// TwinCAT 3 PLC project PRG_Test_Periphery
// Company: RafalOS
// ProgramVersion: 3.1.4024.0
// libraries:
//   B_Actuator, * (RafalOS)
//   B_ActuatorDecorator, * (RafalOS)
//   B_Base, * (RafalOS)
//   B_IO, * (RafalOS)
//   B_IODecorator, * (RafalOS)
//   Tc2_DataExchange, * (Beckhoff Automation GmbH)
//   Tc2_Standard, * (Beckhoff Automation GmbH)
//   Tc2_System, * (Beckhoff Automation GmbH)
//   Tc3_Module, * (Beckhoff Automation GmbH)
//   TcUnit, * (www.tcunit.org)
// project tree:
//   GVLs/ GVL_Actuator.TcGVL, GVL_Decorators.TcGVL, GVL_Variable.TcGVL (not stored)
//   / PlcTask.TcTTO (not stored)
//   POUs/ FB_ActuatorTest.TcPOU, FB_ButtonTest.TcPOU, FB_ElectroValveTest.TcPOU, FB_LampBlinkingTest.TcPOU (not stored), FB_Sensor_DecoratorTestTest.TcPOU, FB_SensorTest.TcPOU (not stored), FB_Actuator_TestDecoratorWithoutTimeTest.TcPOU (not stored), FB_Actuator_TestDecoratorWithTimeTest.TcPOU
//   TESTs/ PRG_Test.TcPOU (not stored)

// ---- GVLs/GVL_Actuator.TcGVL
{attribute 'qualified_only'}
VAR_GLOBAL
	flSS1						: FB_BaseFlag;
	flSTO						: FB_BaseFlag;
	fbLogger					: FB_BaseLogger;
	fbTime						: FB_BaseTime;
	fbLocaciotn					: FB_BaseLocation;	
	stCommonData				: ST_BaseCommonData;

	senActuatorStart			: FB_Sensor_NO;
	senActuatorEnd				: FB_Sensor_NO;
	evActuator					: FB_Electrovalve_5on3_2Coil_Vented;
	
	actActuator					: FB_Actuator (
									senStart	:= senActuatorStart,
	                                senEnd		:= senActuatorEnd,
	                                evControl	:= evActuator
								);
								
END_VAR

// ---- GVLs/GVL_Decorators.TcGVL
{attribute 'qualified_only'}
VAR_GLOBAL
	senNO				: FB_Sensor_NO;
	senNC				: FB_Sensor_NC;
	senNO_2inRow		: FB_Sensor_NO_2InRow;
	
	senNO_TestDecorator			: FB_Sensor_NO_TestDecorator (fbToDecorate := senNO);
	senNC_TestDecorator			: FB_Sensor_NC_TestDecorator (fbToDecorate := senNC);
	senNO_2inRow_TestDecorator	: FB_Sensor_NO_2InRow_TestDecorator (fbToDecorate := senNO_2inRow);
	
	
	senActuator1Start		: FB_Sensor_NO;
	senActuator1End			: FB_Sensor_NO;
	evActuator1				: FB_Electrovalve_5on2_1Coil;

	senActuator1Start_TestCecorator		: FB_Sensor_NO_TestDecorator (fbToDecorate := senActuator1Start);
	senActuator1End_TestDecorator		: FB_Sensor_NO_TestDecorator (fbToDecorate := senActuator1End);
	
	actActuator1			: FB_Actuator (
								senStart	:= senActuator1Start_TestCecorator,
								senEnd		:= senActuator1End_TestDecorator,
								evControl	:= evActuator1
							);
	
	actActuator1_TestWithoutTimeDecorator	: FB_Actuator_TestWithoutTimeDecorator (
											fbToDecorate	:= actActuator1,
											actActuator		:= actActuator1,
											senStart		:= senActuator1Start_TestCecorator,
											senEnd			:= senActuator1End_TestDecorator
										);
	

	actActuator1_TestWithTimeDecorator	: FB_Actuator_TestWithTimeDecorator (
											fbToDecorate	:= actActuator1,
											actActuator		:= actActuator1,
											senStart		:= senActuator1Start_TestCecorator,
											senEnd			:= senActuator1End_TestDecorator
										);
	flSS1						: FB_BaseFlag;
	flSTO						: FB_BaseFlag;
	fbLogger					: FB_BaseLogger;
	fbTime						: FB_BaseTime;
	fbLocaciotn					: FB_BaseLocation;	
	stCommonData				: ST_BaseCommonData;
	
END_VAR

// ---- POUs/FB_ActuatorTest.TcPOU
FUNCTION_BLOCK FB_ActuatorTest EXTENDS TcUnit.FB_TestSuite
VAR

END_VAR


GVL_Actuator.actActuator.ExecuteEveryCycle_Test ();
GVL_Actuator.actActuator.ExecuteEveryCycle_Operation ();
GVL_Actuator.actActuator.ExecuteEveryCycle_Status ();
GVL_Actuator.actActuator.ExecuteEveryCycle_Error ();

T01_Parameter ();
T02_TestMove ();

METHOD PROTECTED T01_Parameter
VAR_INPUT
END_VAR

VAR
	uiWynik: UINT;
	rWynik: REAL;
END_VAR
IF (TcUnit.TEST_ORDERED ('T01_Parameter')) THEN
	GVL_Actuator.stCommonData.itfLocaciotn	:= GVL_Actuator.fbLocaciotn;
	GVL_Actuator.stCommonData.itfLogger		:= GVL_Actuator.fbLogger;
	GVL_Actuator.stCommonData.itfTime		:= GVL_Actuator.fbTime;
	GVL_Actuator.actActuator.LinkCommonData (stCommonData := GVL_Actuator.stCommonData);
	GVL_Actuator.actActuator.LinkSS1 (fbSS1	:= GVL_Actuator.flSS1);
	GVL_Actuator.actActuator.LinkSTO (fbSTO	:= GVL_Actuator.flSTO);
	
	GVL_Actuator.flSS1.SetFlag (bState := TRUE);
	GVL_Actuator.flSTO.SetFlag (bState := TRUE);

	GVL_Actuator.actActuator.ParametersCreate ();
	
	uiWynik		:= GVL_Actuator.actActuator.ParameterGetNumberOfAdded ();
	AssertEquals_UINT (Expected := 2, Actual := uiWynik, Message := 'T01 - Bledna ilosc parametrow');
	rWynik		:= GVL_Actuator.actActuator.ParameterGetValue (uiNumber := 1);
	AssertEquals_REAL (Expected := 100, Actual := rWynik, Delta := 0, Message := 'T02 - bladna wartosc');
	rWynik		:= GVL_Actuator.actActuator.ParameterGetValue (uiNumber := 2);
	AssertEquals_REAL (Expected := 100, Actual := rWynik, Delta := 0, Message := 'T03 - bladna wartosc');

	GVL_Actuator.actActuator.ParameterCorrectValue (uiNumber := 1, rValue := 1000);
	GVL_Actuator.actActuator.ParameterCorrectValue (uiNumber := 2, rValue := 1000);
	rWynik		:= GVL_Actuator.actActuator.ParameterGetValue (uiNumber := 1);
	AssertEquals_REAL (Expected := 1000, Actual := rWynik, Delta := 0, Message := 'T04 - bladna wartosc');
	rWynik		:= GVL_Actuator.actActuator.ParameterGetValue (uiNumber := 2);
	AssertEquals_REAL (Expected := 1000, Actual := rWynik, Delta := 0, Message := 'T05 - bladna wartosc');

	GVL_Actuator.actActuator.ParameterCorrectValue (uiNumber := 1, rValue := 100);
	GVL_Actuator.actActuator.ParameterCorrectValue (uiNumber := 2, rValue := 100);
	
	
	TcUnit.TEST_FINISHED ();
END_IF
END_METHOD

METHOD PRIVATE T02_TestMove
VAR_INST
	iStep			: int;
END_VAR
IF (TcUnit.TEST_ORDERED ('T02_TestMove')) THEN
	CASE iStep OF
	0	:
		GVL_Actuator.actActuator.PowerTurnOn ();
		iStep		:= iStep + 10;
	10	:
		IF (GVL_Actuator.actActuator.PowerTurnOnDone ()) THEN
			iStep	:= iStep + 10;
		END_IF
	20	:
		GVL_Actuator.actActuator.MoveToStart ();
		iStep		:= iStep + 10;
	30	:
		AssertTrue (Condition := GVL_Actuator.actActuator.MovingToStartBusy (), Message := 'S30 - T01 - nie uruchomione przesuwanie');
		AssertFalse (Condition :=GVL_Actuator.actActuator.MovingToStartStatus (), Message := 'S30 - T02 - Bledny status');
		iStep		:= iStep + 10;
	40	:
		GVL_Variable.bValueToSave	:= TRUE;
		GVL_Variable.sData			:= 'GVL_Actuator.senActuatorStart.bContact';
		GVL_Variable.bSave			:= TRUE;
		iStep		:= iStep + 10;
	50	:
		IF (NOT GVL_Variable.bSaved) THEN
			GVL_Variable.bSave		:= FALSE;
			iStep	:= iStep + 10;
		END_IF
	60	:
		AssertFalse (Condition := GVL_Actuator.actActuator.MovingToStartBusy (), Message := 'S60 - T01 - nie zakonczone przesuwanie');
		AssertTrue (Condition := GVL_Actuator.actActuator.MovingToStartStatus (), Message := 'S60 - T02 - Bledny status');
		AssertTrue (Condition := GVL_Actuator.senActuatorStart.IsActive (), Message := 'S60 - T03 - Bledny stan czujnika');
	
		iStep		:= 1000;
	1000	:
		TcUnit.TEST_FINISHED ();
	END_CASE
END_IF
END_METHOD

END_FUNCTION_BLOCK

// ---- POUs/FB_ButtonTest.TcPOU
FUNCTION_BLOCK FB_ButtonTest EXTENDS TcUnit.FB_TestSuite
VAR
END_VAR

T01_Przycisk_NC ();
T02_Przycisk_NO ();
T03_PrzyciskNC_Impuls ();
T04_PrzyciskNO_Impuls ();

METHOD PROTECTED T01_Przycisk_NC
IF (TcUnit.TEST_ORDERED ('T01_Przycisk_NC')) THEN 
	//Przycisk nie jest nacisniety
	WRITE_PROTECTED_BOOL (ADR (GVL_Variable.fbButton_NC.bcontact), TRUE);
	//odczyt
	AssertEquals_BOOL (Actual := GVL_Variable.fbButton_NC.IsPressed (), Expected := FALSE, Message := '1 - Bledny odczyt styku');
	//Przycisk jest nacisniety
	WRITE_PROTECTED_BOOL (ADR (GVL_Variable.fbButton_NC.bContact), FALSE);
	//odczyt
	AssertEquals_BOOL (Actual := GVL_Variable.fbButton_NC.IsPressed (), Expected := TRUE, Message := '2 - Bledny odczyt styku');
	
	TcUnit.TEST_FINISHED ();
END_IF
END_METHOD

METHOD PROTECTED T02_Przycisk_NO
VAR
	bCzyNaciskniety: BOOL;
	bCzySwieci: BOOL;
END_VAR
IF (TcUnit.TEST_ORDERED ('T02_Przycisk_NO')) THEN 
	//Przycisk nie jest nacisniety
	WRITE_PROTECTED_BOOL (ADR (GVL_Variable.fbButton_NO.bContact), FALSE);
	//odczyt
	AssertEquals_BOOL (Actual := GVL_Variable.fbButton_NO.IsPressed (), Expected := FALSE, Message := '1 - Bledny odczyt styku');
	//Przycisk jest nacisniety
	WRITE_PROTECTED_BOOL (ADR (GVL_Variable.fbButton_NO.bContact), TRUE);
	//odczyt
	AssertEquals_BOOL (Actual := GVL_Variable.fbButton_NO.IsPressed (), Expected := TRUE, Message := '2 - Bledny odczyt styku');

	TcUnit.TEST_FINISHED ();
END_IF
END_METHOD

METHOD PROTECTED T03_PrzyciskNC_Impuls
VAR_INST
	iKrok: INT;
END_VAR
IF (TcUnit.TEST_ORDERED ('T03_PrzyciskNC_Impuls')) THEN
	CASE iKrok OF
		0	: 
			WRITE_PROTECTED_BOOL (Ptr := ADR(GVL_Variable.fbButton_NC.bContact), Value := FALSE);
			iKrok		:= 10;
		10	:
			AssertTrue (Condition := GVL_Variable.fbButton_NC.GetRisingEdgePressed (), Message := '10 - Bledny odczyt styku');
			iKrok		:= 20;
		20	:
			AssertFalse (Condition := GVL_Variable.fbButton_NC.GetRisingEdgePressed (), Message := '20 - Bledny odczyt styku');
			iKrok		:= 30;
		30	:
			WRITE_PROTECTED_BOOL (Ptr := ADR(GVL_Variable.fbButton_NC.bContact), Value := TRUE);
			iKrok		:= 40;
		40	:
			AssertFalse (Condition := GVL_Variable.fbButton_NC.GetRisingEdgePressed (), Message := '40 - Bledny odczyt styku');
			iKrok		:= 500;
		500	:
			TcUnit.TEST_FINISHED ();
	END_CASE	
END_IF
END_METHOD

METHOD PROTECTED T04_PrzyciskNO_Impuls
VAR_INST
	iKrok: INT;
END_VAR
IF (TcUnit.TEST_ORDERED ('T04_PrzyciskNO_Impuls')) THEN
	CASE iKrok OF
		0	: 
			WRITE_PROTECTED_BOOL (Ptr := ADR(GVL_Variable.fbButton_NO.bContact), Value := TRUE);
			iKrok		:= 10;
		10	:
			AssertTrue (Condition := GVL_Variable.fbButton_NO.GetRisingEdgePressed (), Message := '10 - Bledny odczyt styku');
			iKrok		:= 20;
		20	:
			AssertFalse (Condition := GVL_Variable.fbButton_NO.GetRisingEdgePressed (), Message := '20 - Bledny odczyt styku');
			iKrok		:= 30;
		30	:
			WRITE_PROTECTED_BOOL (Ptr := ADR(GVL_Variable.fbButton_NO.bContact), Value := FALSE);
			iKrok 		:= 35;
		35	:
			AssertFalse (Condition := GVL_Variable.fbButton_NO.GetRisingEdgePressed (), Message := '35 - Bledny odczyt styku');
			iKrok		:= 40;
		40	:
			WRITE_PROTECTED_BOOL (Ptr := ADR(GVL_Variable.fbButton_NO.bContact), Value := TRUE);
			AssertTrue (Condition := GVL_Variable.fbButton_NO.IsPressed (), Message := '40a - Bledny odczyt styku');
			iKrok 		:= ikrok + 10;
		50	:
			AssertTrue (Condition := GVL_Variable.fbButton_NO.GetRisingEdgePressed (), Message := '50a - Bledny odczyt styku');
			iKrok 		:= ikrok + 10;
		60	:
			AssertFalse (Condition := GVL_Variable.fbButton_NO.GetRisingEdgePressed (), Message := '60b - Bledny odczyt styku');
			iKrok 		:= ikrok + 10;
		70	:
			WRITE_PROTECTED_BOOL (Ptr := ADR(GVL_Variable.fbButton_NO.bContact), Value := FALSE);
			iKrok 		:= ikrok + 10;
		80	:
			AssertFalse (Condition := GVL_Variable.fbButton_NO.GetRisingEdgePressed (), Message := '80c - Bledny odczyt styku');
			iKrok		:= 500;
		500	:
			TcUnit.TEST_FINISHED ();
	END_CASE
	
END_IF
END_METHOD

END_FUNCTION_BLOCK

// ---- POUs/FB_ElectroValveTest.TcPOU
FUNCTION_BLOCK FB_ElectroValveTest EXTENDS TcUnit.FB_TestSuite
VAR
END_VAR

T01_El3Na2_NC ();
T02_El3Na2_NO ();
T03_El5Na2_1C ();
T04_El5Na2_2C ();
T05_El5Na3_2C_odp ();
T06_El5Na3_2C_zap ();

METHOD PROTECTED T01_El3Na2_NC
VAR_INPUT
END_VAR
IF (TcUnit.TEST_ORDERED ('T01_El3Na2_NC')) THEN
	GVL_Variable.ev3on2_NC.Contol (eAction 	:= E_ElectrovalveAction.e_EV_OUT4_Active);
	AssertTrue (
		Condition							:= GVL_Variable.ev3on2_NC.bCoilA,
		Message								:= 'Test 1 - blad przelaczania'
	);
	GVL_Variable.ev3on2_NC.Contol (eAction 	:= E_ElectrovalveAction.e_EV_Out4_Deactive);
	AssertFalse (
		Condition							:= GVL_Variable.ev3on2_NC.bCoilA,
		Message								:= 'Test 2 - blad przelaczania'
	);
	GVL_Variable.ev3on2_NC.Contol (eAction 	:= E_ElectrovalveAction.e_EV_OUT4_Active);
	AssertTrue (
		Condition							:= GVL_Variable.ev3on2_NC.bCoilA,
		Message								:= 'Test 3 - blad przelaczania'
	);
	GVL_Variable.ev3on2_NC.Contol (eAction 	:= E_ElectrovalveAction.e_EV_Reset);
	AssertFalse (
		Condition							:= GVL_Variable.ev3on2_NC.bCoilA,
		Message								:= 'Test 4 - blad przelaczania'
	);
	

	TcUnit.TEST_FINISHED ();
END_IF
END_METHOD

METHOD PROTECTED T02_El3Na2_NO
VAR_INPUT
END_VAR
IF (TcUnit.TEST_ORDERED ('T02_El3Na2_NO')) THEN
	GVL_Variable.ev3on2_NC.Contol (eAction 	:= E_ElectrovalveAction.e_EV_OUT4_Active);
	AssertTrue (
		Condition							:= GVL_Variable.ev3on2_NC.bCoilA,
		Message								:= 'Test 1 - blad przelaczania'
	);
	GVL_Variable.ev3on2_NC.Contol (eAction 	:= E_ElectrovalveAction.e_EV_Out4_Deactive);
	AssertFalse (
		Condition							:= GVL_Variable.ev3on2_NC.bCoilA,
		Message								:= 'Test 2 - blad przelaczania'
	);
	GVL_Variable.ev3on2_NC.Contol (eAction 	:= E_ElectrovalveAction.e_EV_OUT4_Active);
	AssertTrue (
		Condition							:= GVL_Variable.ev3on2_NC.bCoilA,
		Message								:= 'Test 3 - blad przelaczania'
	);
	GVL_Variable.ev3on2_NC.Contol (eAction 	:= E_ElectrovalveAction.e_EV_Reset);
	AssertFalse (
		Condition							:= GVL_Variable.ev3on2_NC.bCoilA,
		Message								:= 'Test 4 - blad przelaczania'
	);
	

	TcUnit.TEST_FINISHED ();
END_IF
END_METHOD

METHOD PROTECTED T03_El5Na2_1C
VAR_INPUT
END_VAR
IF (TcUnit.TEST_ORDERED ('T03_El5Na2_1C')) THEN
	GVL_Variable.ev5on2_1C.Contol (eAction 	:= E_ElectrovalveAction.e_EV_OUT4_Active);
	AssertTrue (
		Condition							:= GVL_Variable.ev5on2_1C.bCoilA,
		Message								:= 'Test 1 - blad przelaczania'
	);
	
	GVL_Variable.ev5on2_1C.Contol (eAction 	:= E_ElectrovalveAction.e_EV_Out4_Deactive);
	AssertFalse (
		Condition							:= GVL_Variable.ev5on2_1C.bCoilA,
		Message								:= 'Test 2 - blad przelaczania'
	);
	
	GVL_Variable.ev5on2_1C.Contol (eAction 	:= E_ElectrovalveAction.e_EV_ToStart);
	AssertFalse (
		Condition							:= GVL_Variable.ev5on2_1C.bCoilA,
		Message								:= 'Test 1 - blad przelaczania'
	);

	GVL_Variable.ev5on2_1C.Contol (eAction 	:= E_ElectrovalveAction.e_EV_ToEnd);
	AssertTrue (
		Condition							:= GVL_Variable.ev5on2_1C.bCoilA,
		Message								:= 'Test 2 - blad przelaczania'
	);
	

	TcUnit.TEST_FINISHED ();
END_IF
END_METHOD

METHOD PROTECTED T04_El5Na2_2C
VAR_INPUT
END_VAR
IF (TcUnit.TEST_ORDERED ('T04_El5Na2_2C')) THEN
	GVL_Variable.ev5on2_2C.Contol (eAction 	:= E_ElectrovalveAction.e_EV_OUT4_Active);
	AssertTrue (
		Condition							:= GVL_Variable.ev5on2_2C.bCoilA,
		Message								:= 'Test 1A - Blad przelaczania'
	);
	Assertfalse (
		Condition							:= GVL_Variable.ev5on2_2C.bCoilB,
		Message								:= 'Test 1B - Blad przelaczania'
	);
//
	GVL_Variable.ev5on2_2C.Contol (eAction 	:= E_ElectrovalveAction.e_EV_Out2_Active);
	AssertFalse (
		Condition							:= GVL_Variable.ev5on2_2C.bCoilA,
		Message								:= 'Test 2A - Blad przelaczania'
	);
	AssertTrue (
		Condition							:= GVL_Variable.ev5on2_2C.bCoilB,
		Message								:= 'Test 2B - Blad przelaczania'
	);
//
	GVL_Variable.ev5on2_2C.Contol (eAction 	:= E_ElectrovalveAction.e_EV_ToEnd);
	AssertTrue (
		Condition							:= GVL_Variable.ev5on2_2C.bCoilA,
		Message								:= 'Test 3A - Blad przelaczania'
	);
	Assertfalse (
		Condition							:= GVL_Variable.ev5on2_2C.bCoilB,
		Message								:= 'Test 3B - Blad przelaczania'
	);
//
	GVL_Variable.ev5on2_2C.Contol (eAction 	:= E_ElectrovalveAction.e_EV_ToStart);
	AssertFalse (
		Condition							:= GVL_Variable.ev5on2_2C.bCoilA,
		Message								:= 'Test 4A - Blad przelaczania'
	);
	AssertTrue (
		Condition							:= GVL_Variable.ev5on2_2C.bCoilB,
		Message								:= 'Test 4B - Blad przelaczania'
	);
//
	GVL_Variable.ev5on2_2C.Contol (eAction 	:= E_ElectrovalveAction.e_EV_Reset);
	AssertFalse (
		Condition							:= GVL_Variable.ev5on2_2C.bCoilA,
		Message								:= 'Test 5A - Blad przelaczania'
	);
	AssertFalse (
		Condition							:= GVL_Variable.ev5on2_2C.bCoilB,
		Message								:= 'Test 5B - Blad przelaczania'
	);
	TcUnit.TEST_FINISHED ();
END_IF
END_METHOD

METHOD PROTECTED T05_El5Na3_2C_odp
VAR_INPUT
END_VAR
IF (TcUnit.TEST_ORDERED ('T05_El5Na3_2C_odp')) THEN
	GVL_Variable.ev5on3_2C_ven.Contol (eAction 	:= E_ElectrovalveAction.e_EV_OUT4_Active);
	AssertTrue (
		Condition							:= GVL_Variable.ev5on3_2C_ven.bCoilA,
		Message								:= 'Test 1A - Blad przelaczania'
	);
//
	GVL_Variable.ev5on3_2C_ven.Contol (eAction 	:= E_ElectrovalveAction.e_EV_Out2_Active);
	AssertTrue (
		Condition							:= GVL_Variable.ev5on3_2C_ven.bCoilB,
		Message								:= 'Test 2B - Blad przelaczania'
	);
//
	GVL_Variable.ev5on3_2C_ven.Contol (eAction 	:= E_ElectrovalveAction.e_EV_Reset);
	AssertFalse (
		Condition							:= GVL_Variable.ev5on3_2C_ven.bCoilA,
		Message								:= 'Test 3A - Blad przelaczania'
	);
	AssertFalse (
		Condition							:= GVL_Variable.ev5on3_2C_ven.bCoilB,
		Message								:= 'Test 3B - Blad przelaczania'
	);
//
	GVL_Variable.ev5on3_2C_ven.Contol (eAction 	:= E_ElectrovalveAction.e_EV_ToStart);
	AssertFalse (
		Condition							:= GVL_Variable.ev5on3_2C_ven.bCoilA,
		Message								:= 'Test 4A - Blad przelaczania'
	);
	AssertTrue (
		Condition							:= GVL_Variable.ev5on3_2C_ven.bCoilB,
		Message								:= 'Test 4B - Blad przelaczania'
	);
//
	GVL_Variable.ev5on3_2C_ven.Contol (eAction 	:= E_ElectrovalveAction.e_EV_ToEnd);
	AssertTrue (
		Condition							:= GVL_Variable.ev5on3_2C_ven.bCoilA,
		Message								:= 'Test 5A - Blad przelaczania'
	);
	Assertfalse (
		Condition							:= GVL_Variable.ev5on3_2C_ven.bCoilB,
		Message								:= 'Test 5B - Blad przelaczania'
	);
//
	GVL_Variable.ev5on3_2C_ven.Contol (eAction 	:= E_ElectrovalveAction.e_EV_Stop);
	AssertTrue (
		Condition							:= GVL_Variable.ev5on3_2C_ven.bCoilA,
		Message								:= 'Test 6A - Blad przelaczania'
	);
	AssertTrue (
		Condition							:= GVL_Variable.ev5on3_2C_ven.bCoilB,
		Message								:= 'Test 6B - Blad przelaczania'
	);
	
	TcUnit.TEST_FINISHED ();
END_IF
END_METHOD

METHOD PROTECTED T06_El5Na3_2C_zap
VAR_INPUT
END_VAR
IF (TcUnit.TEST_ORDERED ('T06_El5Na3_2C_zap')) THEN
	GVL_Variable.ev5on3_2C_inf.Contol (eAction 	:= E_ElectrovalveAction.e_EV_Out4_Deactive);
	AssertTrue (
		Condition							:= GVL_Variable.ev5on3_2C_inf.bCoilA,
		Message								:= 'Test 1A - Blad przelaczania'
	);
//
	GVL_Variable.ev5on3_2C_inf.Contol (eAction 	:= E_ElectrovalveAction.e_EV_Out2_Deactive);
	AssertTrue (
		Condition							:= GVL_Variable.ev5on3_2C_inf.bCoilB,
		Message								:= 'Test 2B - Blad przelaczania'
	);
//
	GVL_Variable.ev5on3_2C_inf.Contol (eAction 	:= E_ElectrovalveAction.e_EV_Reset);
	AssertFalse (
		Condition							:= GVL_Variable.ev5on3_2C_inf.bCoilA,
		Message								:= 'Test 3A - Blad przelaczania'
	);
	AssertFalse (
		Condition							:= GVL_Variable.ev5on3_2C_inf.bCoilB,
		Message								:= 'Test 3B - Blad przelaczania'
	);
//
	GVL_Variable.ev5on3_2C_inf.Contol (eAction 	:= E_ElectrovalveAction.e_EV_ToStart);
	AssertTrue (
		Condition							:= GVL_Variable.ev5on3_2C_inf.bCoilA,
		Message								:= 'Test 4A - Blad przelaczania'
	);
	AssertFalse (
		Condition							:= GVL_Variable.ev5on3_2C_inf.bCoilB,
		Message								:= 'Test 4B - Blad przelaczania'
	);
//
	GVL_Variable.ev5on3_2C_inf.Contol (eAction 	:= E_ElectrovalveAction.e_EV_ToEnd);
	AssertFalse (
		Condition							:= GVL_Variable.ev5on3_2C_inf.bCoilA,
		Message								:= 'Test 5A - Blad przelaczania'
	);
	AssertTrue (
		Condition							:= GVL_Variable.ev5on3_2C_inf.bCoilB,
		Message								:= 'Test 5B - Blad przelaczania'
	);
//
	GVL_Variable.ev5on3_2C_inf.Contol (eAction 	:= E_ElectrovalveAction.e_EV_Stop);
	AssertFalse (
		Condition							:= GVL_Variable.ev5on3_2C_inf.bCoilA,
		Message								:= 'Test 6A - Blad przelaczania'
	);
	AssertFalse (
		Condition							:= GVL_Variable.ev5on3_2C_inf.bCoilB,
		Message								:= 'Test 6B - Blad przelaczania'
	);
	
	TcUnit.TEST_FINISHED ();
END_IF
END_METHOD

END_FUNCTION_BLOCK

// ---- POUs/FB_Sensor_DecoratorTestTest.TcPOU
FUNCTION_BLOCK FB_Sensor_DecoratorTestTest EXTENDS TcUnit.FB_TestSuite
VAR

END_VAR


T01_TestCzujnikNC ();
T02_TestCzujnikNO ();
T03_TestCzujnikNO_Szereg ();

METHOD PROTECTED T01_TestCzujnikNC
VAR_INST
	iKrok		: INT;
END_VAR
IF (TcUnit.TEST_ORDERED ('T01_TestCzujnikNC')) THEN
	GVL_Decorators.senNC_TestDecorator.SetContact (bIN := TRUE);
	AssertFalse (Condition := GVL_Decorators.senNC_TestDecorator.IsActive (), Message := 'T11 - bledny stan');
	GVL_Decorators.senNC_TestDecorator.SetContact (bIN := FALSE);
	AssertTrue (Condition := GVL_Decorators.senNC_TestDecorator.IsActive (), Message := 'T12 - bledny stan');
	GVL_Decorators.senNC_TestDecorator.SetContact (bIN := TRUE);
	AssertFalse (Condition := GVL_Decorators.senNC_TestDecorator.IsActive (), Message := 'T13 - bledny stan');
	
	TcUnit.TEST_FINISHED ();
END_IF
END_METHOD

METHOD PROTECTED T02_TestCzujnikNO
VAR_INST
	iKrok		: INT;
END_VAR
IF (TcUnit.TEST_ORDERED ('T02_TestCzujnikNO')) THEN
	GVL_Decorators.senNO_TestDecorator.SetContact (bIN := FALSE);
	AssertFalse (Condition := GVL_Decorators.senNo_TestDecorator.IsActive (), Message := 'T11 - bledny stan');
	GVL_Decorators.senNO_TestDecorator.SetContact (bIN := TRUE);
	AssertTrue (Condition := GVL_Decorators.senNO_TestDecorator.IsActive (), Message := 'T12 - bledny stan');
	GVL_Decorators.senNO_TestDecorator.SetContact (bIN := FALSE);
	AssertFalse (Condition := GVL_Decorators.senNO_TestDecorator.IsActive (), Message := 'T13 - bledny stan');

	TcUnit.TEST_FINISHED ();
END_IF
END_METHOD

METHOD PROTECTED T03_TestCzujnikNO_Szereg
VAR_INST
	ikrok			: int;
END_VAR
IF (TcUnit.TEST_ORDERED ('T03_TestCzujnikNO_Szereg')) THEN
	GVL_Decorators.senNO_2inRow_TestDecorator.SetContact (bIN := FALSE);
	GVL_Decorators.senNO_2inRow_TestDecorator.SetContact2 (bIN := FALSE);
	AssertFalse (Condition := GVL_Decorators.senNO_2inRow_TestDecorator.IsActive (), Message := 'T11 - bledny stan');
	
	GVL_Decorators.senNO_2inRow_TestDecorator.SetContact (bIN := TRUE);
	AssertFalse (Condition := GVL_Decorators.senNO_2inRow_TestDecorator.IsActive (), Message := 'T12 - bledny stan');

	GVL_Decorators.senNO_2inRow_TestDecorator.SetContact2 (bIN := TRUE);
	AssertTrue (Condition := GVL_Decorators.senNO_2inRow_TestDecorator.IsActive (), Message := 'T13 - bledny stan');

	GVL_Decorators.senNO_2inRow_TestDecorator.SetContact (bIN := FALSE);
	AssertFalse (Condition := GVL_Decorators.senNO_2inRow_TestDecorator.IsActive (), Message := 'T14 - bledny stan');

	GVL_Decorators.senNO_2inRow_TestDecorator.SetContact2 (bIN := FALSE);
	AssertFalse (Condition := GVL_Decorators.senNO_2inRow_TestDecorator.IsActive (), Message := 'T15 - bledny stan');
	
	TcUnit.TEST_FINISHED ();
END_IF
END_METHOD

END_FUNCTION_BLOCK

// ---- POUs/FB_Actuator_TestDecoratorWithTimeTest.TcPOU
FUNCTION_BLOCK INTERNAL FB_Actuator_TestDecoratorWithTimeTest EXTENDS TcUnit.FB_TestSuite
VAR
	uiIlosc					: UINT;	
	tonPrzesuwania			: Tc2_Standard.TON;
	bJest					: BOOL;
	bKoniec					: BOOL;
END_VAR

T00_LinkData ();
GVL_Decorators.actActuator1_TestWithTimeDecorator.ExecuteEveryCycle_Test ();
GVL_Decorators.actActuator1_TestWithTimeDecorator.ExecuteEveryCycle_Operation ();
GVL_Decorators.actActuator1_TestWithTimeDecorator.ExecuteEveryCycle_Status ();
GVL_Decorators.actActuator1_TestWithTimeDecorator.ExecuteEveryCycle_Error ();


T01_TestPracySilownikowWtrybieTestowymDoPoczatku ();
T02_TestPracySilownikowWtrybieTestowymDoKonca ();

T03_TestSilownikaZdekoratoremAutomat ();

METHOD PRIVATE T00_LinkData
VAR_INPUT
END_VAR
IF (TcUnit.TEST_ORDERED ('T00_LinkData')) THEN
	GVL_Decorators.stCommonData.itfLocaciotn	:= GVL_Decorators.fbLocaciotn;
	GVL_Decorators.stCommonData.itfLogger		:= GVL_Decorators.fbLogger;
	GVL_Decorators.stCommonData.itfTime			:= GVL_Decorators.fbTime;
	GVL_Decorators.actActuator1_TestWithTimeDecorator.LinkCommonData (stCommonData := GVL_Decorators.stCommonData);
	GVL_Decorators.actActuator1_TestWithTimeDecorator.LinkSS1 (fbSS1 := GVL_Decorators.flSS1);
	GVL_Decorators.actActuator1_TestWithTimeDecorator.LinkSTO (fbSTO := GVL_Decorators.flSTO);

	GVL_Decorators.flSS1.SetFlag (bState	:= TRUE);
	GVL_Decorators.flSTO.SetFlag (bState	:= TRUE);
	
	GVL_Decorators.actActuator1_TestWithTimeDecorator.ParametersCreate ();

//	uiIlosc	:= GVL_Decorators.fbLogger.

	uiIlosc	:= 1;//fbLoger.ZgloszenieUstawID (uiID 		:= 1);
	GVL_Decorators.actActuator1_TestWithTimeDecorator.SetEventsIDs (uiNewID	:= uiIlosc);
//	fbSilownik_DekoratorTestBezCzasow.ZgloszenieUstawID (uiID	:= uiIlosc);
	
	TcUnit.TEST_FINISHED ();
END_IF
END_METHOD

METHOD PROTECTED T01_TestPracySilownikowWtrybieTestowymDoPoczatku
VAR_INST
	iStep			: INT;
END_VAR
IF (TcUnit.TEST_ORDERED ('T01_TestPracySilownikowWtrybieTestowymDoPoczatku')) THEN
	tonPrzesuwania ();
	CASE iStep OF
	0	:
		GVL_Decorators.actActuator1_TestWithTimeDecorator.PowerTurnOn ();
		iStep	:= 5;
	5	:
		IF (GVL_Decorators.actActuator1_TestWithTimeDecorator.PowerGetStatus ()) THEN
			GVL_Decorators.actActuator1_TestWithTimeDecorator.MoveToStart ();
			tonPrzesuwania.PT			:= REAL_TO_TIME (GVL_Decorators.actActuator1_TestWithTimeDecorator.ParameterGetValue (uiNumber := 1)*0.25);
			tonPrzesuwania.IN			:= TRUE;
			iStep						:= iStep + 5;
		END_IF
	10	:
		IF (tonPrzesuwania.Q) THEN
			tonPrzesuwania.IN		:= FALSE;
			AssertFalse (Condition	:= GVL_Decorators.actActuator1_TestWithTimeDecorator.MovingToStartStatus (),Message 	:= 'K10 T01 - czy juz dojechal');
			AssertTrue (Condition	:= GVL_Decorators.actActuator1_TestWithTimeDecorator.MovingToStartBusy (), 	Message 	:= 'K10 T02 - nie wlaczono przesuwania');
			iStep					:= iStep + 10;
		END_IF
	20	:
		tonPrzesuwania.PT			:= REAL_TO_TIME (GVL_Decorators.actActuator1_TestWithTimeDecorator.ParameterGetValue (uiNumber := 1)*0.75);
		tonPrzesuwania.IN			:= TRUE;
		iStep						:= iStep + 10;
	30	:
		IF (tonPrzesuwania.Q) THEN
			tonPrzesuwania.IN		:= FALSE;
			AssertTrue (Condition	:= GVL_Decorators.actActuator1_TestWithTimeDecorator.MovingToStartStatus (),Message 	:= 'K30 T01 - czy juz dojechal');
			AssertFalse (Condition	:= GVL_Decorators.actActuator1_TestWithTimeDecorator.MovingToStartBusy (), 	Message 	:= 'K30 T02 - nie wlaczono przesuwania');
			iStep					:= iStep + 10;
		END_IF
	40	:
		iStep	:= GVL_BaseConstans.FINISH_STEP;
	GVL_BaseConstans.FINISH_STEP	:
		TcUnit.TEST_FINISHED ();
	END_CASE

END_IF
END_METHOD

METHOD PROTECTED T02_TestPracySilownikowWtrybieTestowymDoKonca
VAR_INST
	iStep			: INT;
END_VAR
IF (TcUnit.TEST_ORDERED ('T02_TestPracySilownikowWtrybieTestowymDoKonca')) THEN
	tonPrzesuwania ();
	CASE iStep OF
	0	:
		GVL_Decorators.actActuator1_TestWithTimeDecorator.PowerTurnOn ();
		iStep		:= 5;
	5	:
		IF (GVL_Decorators.actActuator1_TestWithTimeDecorator.PowerGetStatus ()) THEN
			GVL_Decorators.actActuator1_TestWithTimeDecorator.MoveToEnd ();
			tonPrzesuwania.PT			:= REAL_TO_TIME (GVL_Decorators.actActuator1_TestWithTimeDecorator.ParameterGetValue(uiNumber := 2)*0.25);
			tonPrzesuwania.IN			:= TRUE;
			iStep						:= iStep + 5;
		END_IF
	10	:
		IF (tonPrzesuwania.Q) THEN
			tonPrzesuwania.IN		:= FALSE;
			AssertFalse (Condition	:= GVL_Decorators.actActuator1_TestWithTimeDecorator.MovingToEndStatus (),	Message 	:= 'K10 T01 - czy juz dojechal');
			AssertTrue (Condition	:= GVL_Decorators.actActuator1_TestWithTimeDecorator.MovingToEndBusy (), 	Message 	:= 'K10 T02 - nie wlaczono przesuwania');
			iStep					:= iStep + 10;
		END_IF
	20	:
		tonPrzesuwania.PT			:= REAL_TO_TIME (GVL_Decorators.actActuator1_TestWithTimeDecorator.ParameterGetValue (uiNumber := 2)*0.75);
		tonPrzesuwania.IN			:= TRUE;
		iStep						:= iStep + 10;
	30	:
		IF (tonPrzesuwania.Q) THEN
			tonPrzesuwania.IN		:= FALSE;
			AssertTrue (Condition	:= GVL_Decorators.actActuator1_TestWithTimeDecorator.MovingToEndStatus (),	Message 	:= 'K30 T01 - czy juz dojechal');
			AssertFalse (Condition	:= GVL_Decorators.actActuator1_TestWithTimeDecorator.MovingToEndBusy (), 	Message 	:= 'K30 T02 - nie wlaczono przesuwania');
			iStep					:= iStep + 10;
		END_IF
	40	:
		iStep	:= GVL_BaseConstans.FINISH_STEP;
	GVL_BaseConstans.FINISH_STEP	:
		TcUnit.TEST_FINISHED ();
	END_CASE

END_IF
END_METHOD

METHOD PROTECTED T03_TestSilownikaZdekoratoremAutomat
VAR_INPUT
END_VAR
IF (TcUnit.TEST_ORDERED ('T03_TestSilownikaZdekoratoremAutomat')) THEN
	bJest			:= TRUE;
	IF (bKoniec) THEN
		bJest		:= FALSE;
		TcUnit.TEST_FINISHED ();
	END_IF
END_IF
END_METHOD

END_FUNCTION_BLOCK
